FUNCTION_BLOCK METHOD_CALLER
  {SET_ATTRIBUTE(OpcUa, SERVICE)}
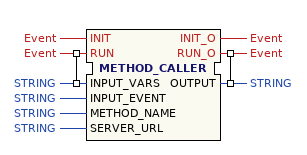
  EVENT_INPUT
    INIT;
    RUN WITH INPUT_VARS;
  END_EVENT
  EVENT_OUTPUT
    INIT_O;
    RUN_O WITH OUTPUT;
  END_EVENT
  VAR_INPUT
    INPUT_VARS : STRING; {SET_ATTRIBUTE(OpcUa, Constant.INIT)}
    INPUT_EVENT : STRING; {SET_ATTRIBUTE(OpcUa, Constant.INIT)}
    METHOD_NAME : STRING; {SET_ATTRIBUTE(OpcUa, Constant.INIT)}
    SERVER_URL : STRING; {SET_ATTRIBUTE(OpcUa, Constant.INIT)}
  END_VAR
  VAR_OUTPUT
    OUTPUT : STRING; {SET_ATTRIBUTE(OpcUa, Constant.INIT)}
  END_VAR
END_FUNCTION_BLOCK
